// TIA Portal V15 export
FUNCTION "PresetStoreEnabled" : Void   // FC30, SCL
{ S7_Optimized_Access := 'TRUE' }
VERSION : 0.1
// stored: AutoNumber true, IsIECCheckEnabled false, SetENOAutomatically False
   VAR_INPUT
      Enable : "PresetEnableType";
   END_VAR
   VAR_OUTPUT
      Value : "PresetValueType";
   END_VAR
BEGIN
END_FUNCTION
